# EPICS substitutions: l2MpsAsynApp/Db/mps_blm.substitutions
### Threshold information ###
file "RegRO.template" { pattern
{ R,                DESC,                                               PARAM,                  ADDR        }
{ I0_THR_CH,        "Bay $(BAY) Ch $(INP) Int 0 Threshold channel",     BLM_THRNUM_$(INP)0,     "$(BAY)"    }
{ I0_THR_CNT,       "Bay $(BAY) Ch $(INP) Int 0 Threshold count",       BLM_THRCNT_$(INP)0,     "$(BAY)"    }
{ I0_THR_BYTEMAP,   "Bay $(BAY) Ch $(INP) Int 0 Threshold byte map",    BLM_BYTEMAP_$(INP)0,    "$(BAY)"    }
}

### Tables enable PVs ###
file "Reg1BitRW.template" { pattern
{ R,                DESC,                                               PARAM,                  ADDR,       ZNAM,           ONAM,      }
{ I0_IDL_EN,        "Bay $(BAY) Ch $(INP) Int 0 IDLE table enabled",    BLM_IDLEEN_$(INP)0,     "$(BAY)",   "Disabled",     "Enabled"  }
}

file "Reg1BitRO.template" { pattern
{ R,                DESC,                                               PARAM,                  ADDR,       ZNAM,           ONAM,      }
{ I0_ALT_EN,        "Bay $(BAY) Ch $(INP) Int 0 ALT table enabled",     BLM_ALTEN_$(INP)0,      "$(BAY)",   "Disabled",     "Enabled"  }
{ I0_LC1_EN,        "Bay $(BAY) Ch $(INP) Int 0 LCLS1 table enabled",   BLM_LCLS1EN_$(INP)0,    "$(BAY)",   "Disabled",     "Enabled"  }
}

### Threshold PVs ###
file "thr.template" { pattern
{ R,                DESC,                                               APP,        EGU,    PREC,   CH,           TABLE,  THR,    }
{ I0_T0_LC1,        "Bay $(BAY) Ch $(INP) Int 0 LCLS1, Threshold",      "BLM",      "",     "2",    "$(INP)0",    "0",    "0",    }

{ I0_T0_IDL,        "Bay $(BAY) Ch $(INP) Int 0 IDLE, Threshold",       "BLM",      "",     "2",    "$(INP)0",    "1",    "0",    }

{ I0_T0,            "Bay $(BAY) Ch $(INP) Int 0 STD, Threshold 0",      "BLM",      "",     "2",    "$(INP)0",    "2",    "0",    }
{ I0_T1,            "Bay $(BAY) Ch $(INP) Int 0 STD, Threshold 1",      "BLM",      "",     "2",    "$(INP)0",    "2",    "1",    }
{ I0_T2,            "Bay $(BAY) Ch $(INP) Int 0 STD, Threshold 2",      "BLM",      "",     "2",    "$(INP)0",    "2",    "2",    }
{ I0_T3,            "Bay $(BAY) Ch $(INP) Int 0 STD, Threshold 3",      "BLM",      "",     "2",    "$(INP)0",    "2",    "3",    }
{ I0_T4,            "Bay $(BAY) Ch $(INP) Int 0 STD, Threshold 4",      "BLM",      "",     "2",    "$(INP)0",    "2",    "4",    }
{ I0_T5,            "Bay $(BAY) Ch $(INP) Int 0 STD, Threshold 5",      "BLM",      "",     "2",    "$(INP)0",    "2",    "5",    }
{ I0_T6,            "Bay $(BAY) Ch $(INP) Int 0 STD, Threshold 6",      "BLM",      "",     "2",    "$(INP)0",    "2",    "6",    }
{ I0_T7,            "Bay $(BAY) Ch $(INP) Int 0 STD, Threshold 7",      "BLM",      "",     "2",    "$(INP)0",    "2",    "7",    }

{ I0_T0_ALT,        "Bay $(BAY) Ch $(INP) Int 0 ALT, Threshold 0",      "BLM",      "",     "2",    "$(INP)0",    "3",    "0",    }
{ I0_T1_ALT,        "Bay $(BAY) Ch $(INP) Int 0 ALT, Threshold 1",      "BLM",      "",     "2",    "$(INP)0",    "3",    "1",    }
{ I0_T2_ALT,        "Bay $(BAY) Ch $(INP) Int 0 ALT, Threshold 2",      "BLM",      "",     "2",    "$(INP)0",    "3",    "2",    }
{ I0_T3_ALT,        "Bay $(BAY) Ch $(INP) Int 0 ALT, Threshold 3",      "BLM",      "",     "2",    "$(INP)0",    "3",    "3",    }
{ I0_T4_ALT,        "Bay $(BAY) Ch $(INP) Int 0 ALT, Threshold 4",      "BLM",      "",     "2",    "$(INP)0",    "3",    "4",    }
{ I0_T5_ALT,        "Bay $(BAY) Ch $(INP) Int 0 ALT, Threshold 5",      "BLM",      "",     "2",    "$(INP)0",    "3",    "5",    }
{ I0_T6_ALT,        "Bay $(BAY) Ch $(INP) Int 0 ALT, Threshold 6",      "BLM",      "",     "2",    "$(INP)0",    "3",    "6",    }
{ I0_T7_ALT,        "Bay $(BAY) Ch $(INP) Int 0 ALT, Threshold 7",      "BLM",      "",     "2",    "$(INP)0",    "3",    "7",    }
}

### Scale PVs ###
file "scale.template" { pattern
{ R,                DESC,                                   APP,        EGU,    PREC,       CH,           SCALE_SLOPE_PV,   SCALE_OFFSET_PV,    SCAN        }
{ I0,               "Bay $(BAY) Ch $(INP) Int 0 Scale ",    "BLM",      "A",    "4",        "$(INP)0",    "$(P):I0_FWSLO",  "$(P):I0_FWOFF",    "1 second"  }
}
